// TIA Portal project "Buffer" (V18)

(* hardware
DEVICE "S7-1500/ET200MP station_1"  S7-1500 station
   slot 0: "Rail_0"  Rack  6ES7 590-1***0-0AA0
   slot 1: "PLC_1"  CPU 1515-2 PN  6ES7 515-2AN03-0AB0  V3.0
      slot 3: "CPU display_1"  6ES7591-1BA00-0AA0
      slot 32768: "PROFINET interface_1"  X1
         slot 32769: "Port_1"  X1 P1
         slot 32770: "Port_2"  X1 P2
      slot 33024: "PROFINET interface_2"  X2
         slot 33025: "Port_1"  X2 P1
      slot 34817: "Virtual CP interface port_1"  Virtual CP interface port  Virtual CP interface port
*)

// ===== PLC "PLC_1"  CPU 1515-2 PN =====

VAR_GLOBAL   // PLC tag table "Default tag table"
   "System_Byte" AT %MB0 : Byte;
   "FirstScan" AT %M0.0 : Bool;
   "DiagStatusUpdate" AT %M0.1 : Bool;
   "AlwaysTRUE" AT %M0.2 : Bool;
   "AlwaysFALSE" AT %M0.3 : Bool;
   "Clock_Byte" AT %MB1 : Byte;
   "Clock_10Hz" AT %M1.0 : Bool;
   "Clock_5Hz" AT %M1.1 : Bool;
   "Clock_2.5Hz" AT %M1.2 : Bool;
   "Clock_2Hz" AT %M1.3 : Bool;
   "Clock_1.25Hz" AT %M1.4 : Bool;
   "Clock_1Hz" AT %M1.5 : Bool;
   "Clock_0.625Hz" AT %M1.6 : Bool;
   "Clock_0.5Hz" AT %M1.7 : Bool;
   "Index" AT %MD18 : UDInt;
   "Start" AT %M16.0 : Bool;
   "Start2" AT %M16.1 : Bool;
   "FoundIndex" AT %MW20 : Word;
   "Tag_1" AT %M16.2 : Bool;
   "Tag_2" AT %MW22 : Int;
END_VAR

VAR_GLOBAL CONSTANT   // PLC tag table "Default tag table"
   "c_MAX_RECORD_LEN" : Int := 100;   // //Max length of single record [Byte]
END_VAR

TYPE "udt_DATABASE3"
   STRUCT
      FirstName : Array[1..10] of Char;
      Lastname : Array[1..20] of Char;
      Age : USInt;
      Details : Struct
         Male : Bool;
         COMPLETE_TO_WORD2 : Bool;
         COMPLETE_TO_WORD3 : Bool;
         COMPLETE_TO_WORD4 : Bool;
         COMPLETE_TO_WORD5 : Bool;
         COMPLETE_TO_WORD6 : Bool;
         COMPLETE_TO_WORD7 : Bool;
         COMPLETE_TO_WORD8 : Bool;
         COMPLETE_TO_WORD9 : Bool;
         COMPLETE_TO_WORD10 : Bool;
         COMPLETE_TO_WORD11 : Bool;
         COMPLETE_TO_WORD12 : Bool;
         COMPLETE_TO_WORD13 : Bool;
         COMPLETE_TO_WORD14 : Bool;
         COMPLETE_TO_WORD15 : Bool;
         COMPLETE_TO_WORD16 : Bool;
      END_STRUCT;
   END_STRUCT;
END_TYPE

// folder: DATABASES

DATA_BLOCK "db_DATABASE_1"   // DB100
{ S7_Optimized_Access := 'TRUE' }
VERSION : 0.1
   VAR
      Act_Records : UDInt;
      WorkRecord : Byte;
      RecordMask : Byte;
      Database : Array[1..1000] of Byte;
   END_VAR
BEGIN
END_DATA_BLOCK

DATA_BLOCK "db_DATABASE_2"   // DB101
{ S7_Optimized_Access := 'TRUE' }
VERSION : 0.1
   VAR
      Act_Records : UDInt;
      WorkRecord : Real;
      RecordMask : Real;
      Database : Array[1..1000] of Real;
   END_VAR
BEGIN
END_DATA_BLOCK

DATA_BLOCK "db_DATABASE_3"   // DB102
{ S7_Optimized_Access := 'TRUE' }
VERSION : 0.1
   VAR
      Act_Records : UDInt;
      WorkRecord : "udt_DATABASE3";
      RecordMask : "udt_DATABASE3";
      Database : Array[1..1000] of "udt_DATABASE3";
   END_VAR
BEGIN
END_DATA_BLOCK

// folder: DB_TOOLS

DATA_BLOCK "db_Records"   // DB1
{ S7_Optimized_Access := 'TRUE' }
VERSION : 0.1
   VAR
      Push : Struct
         Record1 : Byte;
         Record2 : Real;
         Record3 : "udt_DATABASE3";
      END_STRUCT;
      Pop : Struct
         Record1 : Byte;
         Record2 : Real;
         Record3 : "udt_DATABASE3";
      END_STRUCT;
      Shift : Struct
         Record1 : Byte;
         Record2 : Real;
         Record3 : "udt_DATABASE3";
      END_STRUCT;
      Unshift : Struct
         Record1 : Byte;
         Record2 : Real;
         Record3 : "udt_DATABASE3";
      END_STRUCT;
      Insert : Struct
         Record1 : Byte;
         Record2 : Real;
         Record3 : "udt_DATABASE3";
      END_STRUCT;
      Remove : Struct
         Record1 : Byte;
         Record2 : Real;
         Record3 : "udt_DATABASE3";
      END_STRUCT;
      Read : Struct
         Record1 : Byte;
         Record2 : Real;
         Record3 : "udt_DATABASE3";
      END_STRUCT;
      ReadLast : Struct
         Record1 : Byte;
         Record2 : Real;
         Record3 : "udt_DATABASE3";
      END_STRUCT;
      Overwrite : Struct
         Record1 : Byte;
         Record2 : Real;
         Record3 : "udt_DATABASE3";
      END_STRUCT;
      OverwriteLast : Struct
         Record1 : Byte;
         Record2 : Real;
         Record3 : "udt_DATABASE3";
      END_STRUCT;
      Find : Struct
         Record1 : Byte;
         Record2 : Real;
         Record3 : "udt_DATABASE3";
      END_STRUCT;
   END_VAR
BEGIN
END_DATA_BLOCK

// folder: (top level)

FUNCTION "fc_PushCall" : Void   // FC1, LAD
{ S7_Optimized_Access := 'TRUE' }
VERSION : 0.1
   VAR_TEMP
      _DONE : Bool;
   END_VAR
BEGIN

REGION Network 1: Push into Database 1
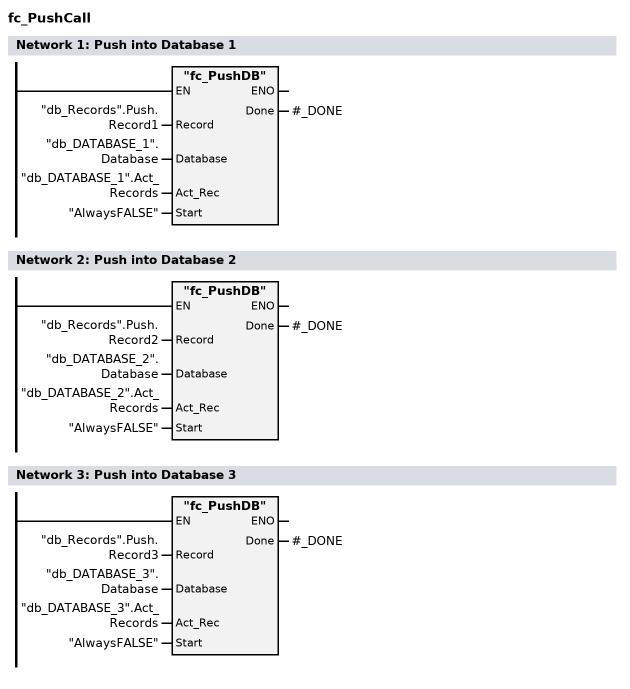
   RUNG wire#powerrail
      "fc_PushDB"(Record := "db_Records".Push.Record1, Database := "db_DATABASE_1".Database, Act_Rec := "db_DATABASE_1".Act_Records, Start := "AlwaysFALSE", Done => #_DONE)
   END_RUNG
   // the same network as SCL:
   "fc_PushDB"(Record := "db_Records".Push.Record1,
               Database := "db_DATABASE_1".Database,
               Act_Rec := "db_DATABASE_1".Act_Records,
               Start := "AlwaysFALSE",
               Done => #_DONE);
END_REGION

REGION Network 2: Push into Database 2
   RUNG wire#powerrail
      "fc_PushDB"(Record := "db_Records".Push.Record2, Database := "db_DATABASE_2".Database, Act_Rec := "db_DATABASE_2".Act_Records, Start := "AlwaysFALSE", Done => #_DONE)
   END_RUNG
   // the same network as SCL:
   "fc_PushDB"(Record := "db_Records".Push.Record2,
               Database := "db_DATABASE_2".Database,
               Act_Rec := "db_DATABASE_2".Act_Records,
               Start := "AlwaysFALSE",
               Done => #_DONE);
END_REGION

REGION Network 3: Push into Database 3
   RUNG wire#powerrail
      "fc_PushDB"(Record := "db_Records".Push.Record3, Database := "db_DATABASE_3".Database, Act_Rec := "db_DATABASE_3".Act_Records, Start := "AlwaysFALSE", Done => #_DONE)
   END_RUNG
   // the same network as SCL:
   "fc_PushDB"(Record := "db_Records".Push.Record3,
               Database := "db_DATABASE_3".Database,
               Act_Rec := "db_DATABASE_3".Act_Records,
               Start := "AlwaysFALSE",
               Done => #_DONE);
END_REGION
END_FUNCTION

FUNCTION "fc_PopCall" : Void   // FC2, LAD
{ S7_Optimized_Access := 'TRUE' }
VERSION : 0.1
   VAR_TEMP
      _DONE : Bool;
   END_VAR
BEGIN

REGION Network 1: Pop from Database 1
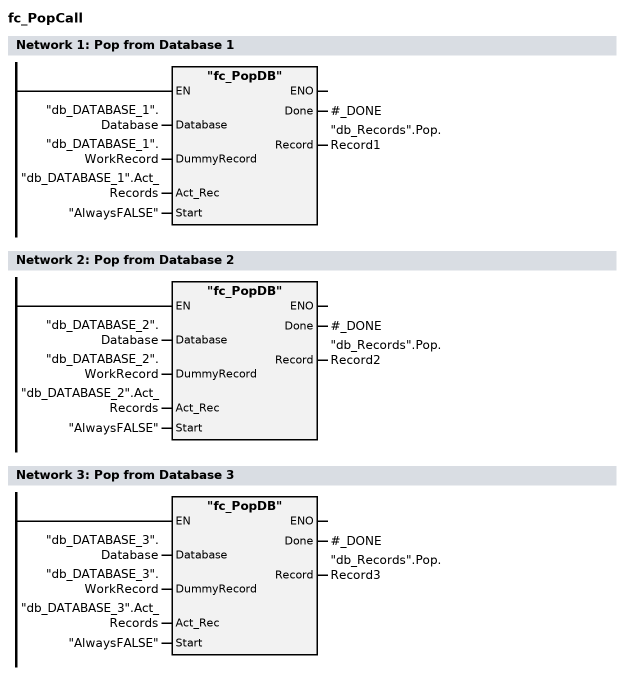
   RUNG wire#powerrail
      "fc_PopDB"(Database := "db_DATABASE_1".Database, DummyRecord := "db_DATABASE_1".WorkRecord, Act_Rec := "db_DATABASE_1".Act_Records, Start := "AlwaysFALSE", Done => #_DONE, Record => "db_Records".Pop.Record1)
   END_RUNG
   // the same network as SCL:
   "fc_PopDB"(Database := "db_DATABASE_1".Database,
              DummyRecord := "db_DATABASE_1".WorkRecord,
              Act_Rec := "db_DATABASE_1".Act_Records,
              Start := "AlwaysFALSE",
              Done => #_DONE,
              Record => "db_Records".Pop.Record1);
END_REGION

REGION Network 2: Pop from Database 2
   RUNG wire#powerrail
      "fc_PopDB"(Database := "db_DATABASE_2".Database, DummyRecord := "db_DATABASE_2".WorkRecord, Act_Rec := "db_DATABASE_2".Act_Records, Start := "AlwaysFALSE", Done => #_DONE, Record => "db_Records".Pop.Record2)
   END_RUNG
   // the same network as SCL:
   "fc_PopDB"(Database := "db_DATABASE_2".Database,
              DummyRecord := "db_DATABASE_2".WorkRecord,
              Act_Rec := "db_DATABASE_2".Act_Records,
              Start := "AlwaysFALSE",
              Done => #_DONE,
              Record => "db_Records".Pop.Record2);
END_REGION

REGION Network 3: Pop from Database 3
   RUNG wire#powerrail
      "fc_PopDB"(Database := "db_DATABASE_3".Database, DummyRecord := "db_DATABASE_3".WorkRecord, Act_Rec := "db_DATABASE_3".Act_Records, Start := "AlwaysFALSE", Done => #_DONE, Record => "db_Records".Pop.Record3)
   END_RUNG
   // the same network as SCL:
   "fc_PopDB"(Database := "db_DATABASE_3".Database,
              DummyRecord := "db_DATABASE_3".WorkRecord,
              Act_Rec := "db_DATABASE_3".Act_Records,
              Start := "AlwaysFALSE",
              Done => #_DONE,
              Record => "db_Records".Pop.Record3);
END_REGION
END_FUNCTION

FUNCTION "fc_ShiftCall" : Void   // FC3, LAD
{ S7_Optimized_Access := 'TRUE' }
VERSION : 0.1
   VAR_TEMP
      _DONE : Bool;
   END_VAR
BEGIN

REGION Network 1: Shift from Database 1
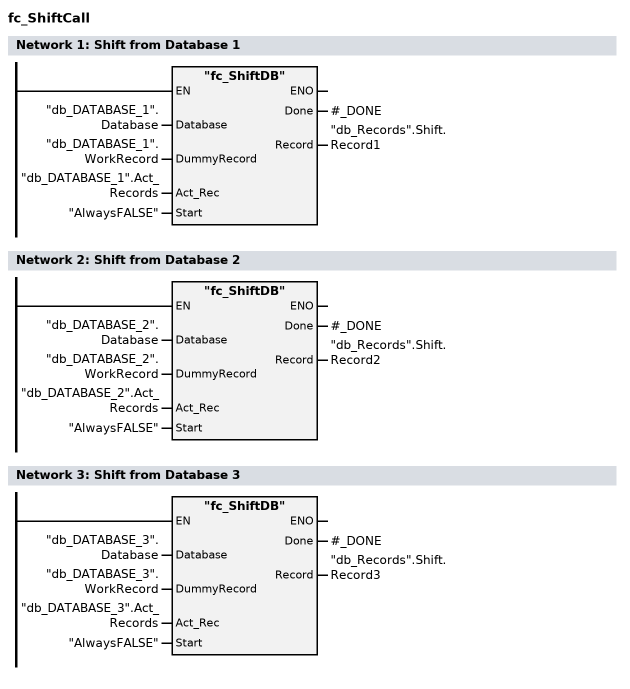
   RUNG wire#powerrail
      "fc_ShiftDB"(Record => "db_Records".Shift.Record1, Database := "db_DATABASE_1".Database, DummyRecord := "db_DATABASE_1".WorkRecord, Act_Rec := "db_DATABASE_1".Act_Records, Start := "AlwaysFALSE", Done => #_DONE)
   END_RUNG
   // the same network as SCL:
   "fc_ShiftDB"(Database := "db_DATABASE_1".Database,
                DummyRecord := "db_DATABASE_1".WorkRecord,
                Act_Rec := "db_DATABASE_1".Act_Records,
                Start := "AlwaysFALSE",
                Done => #_DONE,
                Record => "db_Records".Shift.Record1);
END_REGION

REGION Network 2: Shift from Database 2
   RUNG wire#powerrail
      "fc_ShiftDB"(Record => "db_Records".Shift.Record2, Database := "db_DATABASE_2".Database, DummyRecord := "db_DATABASE_2".WorkRecord, Act_Rec := "db_DATABASE_2".Act_Records, Start := "AlwaysFALSE", Done => #_DONE)
   END_RUNG
   // the same network as SCL:
   "fc_ShiftDB"(Database := "db_DATABASE_2".Database,
                DummyRecord := "db_DATABASE_2".WorkRecord,
                Act_Rec := "db_DATABASE_2".Act_Records,
                Start := "AlwaysFALSE",
                Done => #_DONE,
                Record => "db_Records".Shift.Record2);
END_REGION

REGION Network 3: Shift from Database 3
   RUNG wire#powerrail
      "fc_ShiftDB"(Record => "db_Records".Shift.Record3, Database := "db_DATABASE_3".Database, DummyRecord := "db_DATABASE_3".WorkRecord, Act_Rec := "db_DATABASE_3".Act_Records, Start := "AlwaysFALSE", Done => #_DONE)
   END_RUNG
   // the same network as SCL:
   "fc_ShiftDB"(Database := "db_DATABASE_3".Database,
                DummyRecord := "db_DATABASE_3".WorkRecord,
                Act_Rec := "db_DATABASE_3".Act_Records,
                Start := "AlwaysFALSE",
                Done => #_DONE,
                Record => "db_Records".Shift.Record3);
END_REGION
END_FUNCTION

FUNCTION "fc_UnshiftCall" : Void   // FC4, LAD
{ S7_Optimized_Access := 'TRUE' }
VERSION : 0.1
   VAR_TEMP
      _DONE : Bool;
   END_VAR
BEGIN

REGION Network 1: Unshift into Database 1
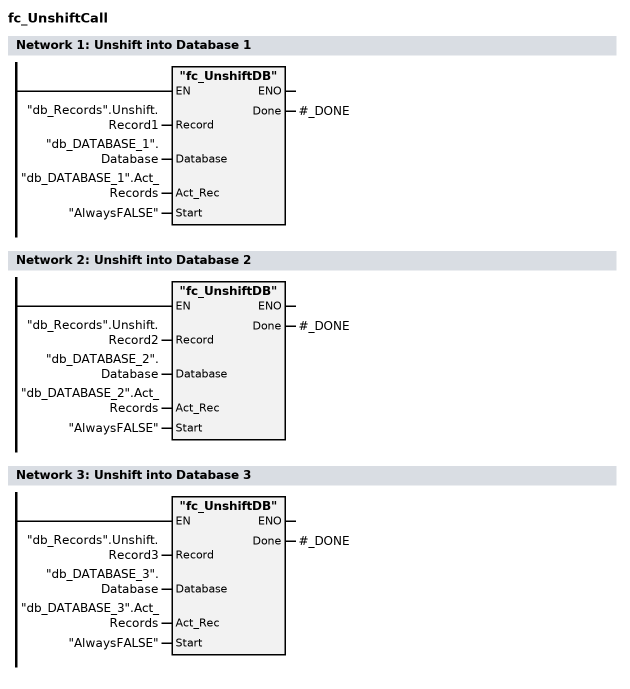
   RUNG wire#powerrail
      "fc_UnshiftDB"(Record := "db_Records".Unshift.Record1, Database := "db_DATABASE_1".Database, Act_Rec := "db_DATABASE_1".Act_Records, Start := "AlwaysFALSE", Done => #_DONE)
   END_RUNG
   // the same network as SCL:
   "fc_UnshiftDB"(Record := "db_Records".Unshift.Record1,
                  Database := "db_DATABASE_1".Database,
                  Act_Rec := "db_DATABASE_1".Act_Records,
                  Start := "AlwaysFALSE",
                  Done => #_DONE);
END_REGION

REGION Network 2: Unshift into Database 2
   RUNG wire#powerrail
      "fc_UnshiftDB"(Record := "db_Records".Unshift.Record2, Database := "db_DATABASE_2".Database, Act_Rec := "db_DATABASE_2".Act_Records, Start := "AlwaysFALSE", Done => #_DONE)
   END_RUNG
   // the same network as SCL:
   "fc_UnshiftDB"(Record := "db_Records".Unshift.Record2,
                  Database := "db_DATABASE_2".Database,
                  Act_Rec := "db_DATABASE_2".Act_Records,
                  Start := "AlwaysFALSE",
                  Done => #_DONE);
END_REGION

REGION Network 3: Unshift into Database 3
   RUNG wire#powerrail
      "fc_UnshiftDB"(Record := "db_Records".Unshift.Record3, Database := "db_DATABASE_3".Database, Act_Rec := "db_DATABASE_3".Act_Records, Start := "AlwaysFALSE", Done => #_DONE)
   END_RUNG
   // the same network as SCL:
   "fc_UnshiftDB"(Record := "db_Records".Unshift.Record3,
                  Database := "db_DATABASE_3".Database,
                  Act_Rec := "db_DATABASE_3".Act_Records,
                  Start := "AlwaysFALSE",
                  Done => #_DONE);
END_REGION
END_FUNCTION

FUNCTION "fc_ClearCall" : Void   // FC5, LAD
{ S7_Optimized_Access := 'TRUE' }
VERSION : 0.1
   VAR_TEMP
      _DONE : Bool;
   END_VAR
BEGIN

REGION Network 1: Clear Database 1
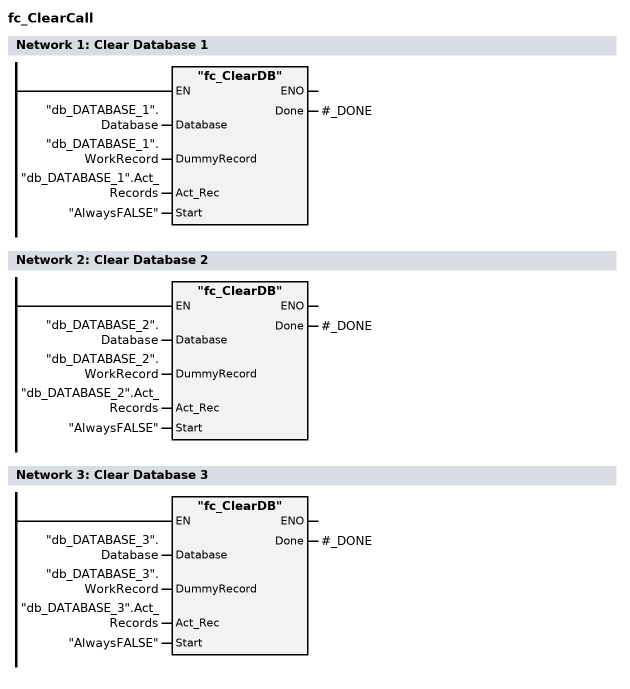
   RUNG wire#powerrail
      "fc_ClearDB"(Database := "db_DATABASE_1".Database, DummyRecord := "db_DATABASE_1".WorkRecord, Act_Rec := "db_DATABASE_1".Act_Records, Start := "AlwaysFALSE", Done => #_DONE)
   END_RUNG
   // the same network as SCL:
   "fc_ClearDB"(Database := "db_DATABASE_1".Database,
                DummyRecord := "db_DATABASE_1".WorkRecord,
                Act_Rec := "db_DATABASE_1".Act_Records,
                Start := "AlwaysFALSE",
                Done => #_DONE);
END_REGION

REGION Network 2: Clear Database 2
   RUNG wire#powerrail
      "fc_ClearDB"(Database := "db_DATABASE_2".Database, DummyRecord := "db_DATABASE_2".WorkRecord, Act_Rec := "db_DATABASE_2".Act_Records, Start := "AlwaysFALSE", Done => #_DONE)
   END_RUNG
   // the same network as SCL:
   "fc_ClearDB"(Database := "db_DATABASE_2".Database,
                DummyRecord := "db_DATABASE_2".WorkRecord,
                Act_Rec := "db_DATABASE_2".Act_Records,
                Start := "AlwaysFALSE",
                Done => #_DONE);
END_REGION

REGION Network 3: Clear Database 3
   RUNG wire#powerrail
      "fc_ClearDB"(Database := "db_DATABASE_3".Database, DummyRecord := "db_DATABASE_3".WorkRecord, Act_Rec := "db_DATABASE_3".Act_Records, Start := "AlwaysFALSE", Done => #_DONE)
   END_RUNG
   // the same network as SCL:
   "fc_ClearDB"(Database := "db_DATABASE_3".Database,
                DummyRecord := "db_DATABASE_3".WorkRecord,
                Act_Rec := "db_DATABASE_3".Act_Records,
                Start := "AlwaysFALSE",
                Done => #_DONE);
END_REGION
END_FUNCTION

FUNCTION "fc_InsertCall" : Void   // FC6, LAD
{ S7_Optimized_Access := 'TRUE' }
VERSION : 0.1
   VAR_TEMP
      _DONE : Bool;
   END_VAR
BEGIN

REGION Network 1: Insert into Database 1
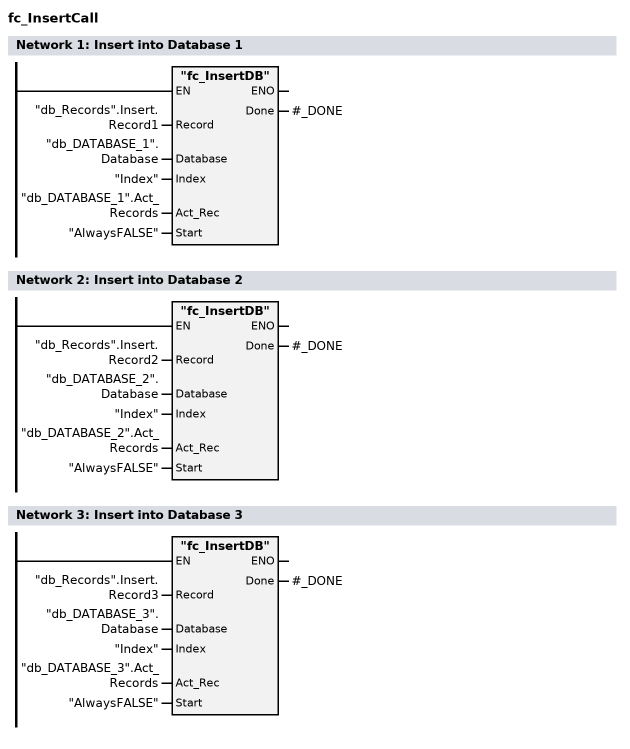
   RUNG wire#powerrail
      "fc_InsertDB"(Record := "db_Records".Insert.Record1, Database := "db_DATABASE_1".Database, Index := "Index", Act_Rec := "db_DATABASE_1".Act_Records, Start := "AlwaysFALSE", Done => #_DONE)
   END_RUNG
   // the same network as SCL:
   "fc_InsertDB"(Record := "db_Records".Insert.Record1,
                 Database := "db_DATABASE_1".Database,
                 Index := "Index",
                 Act_Rec := "db_DATABASE_1".Act_Records,
                 Start := "AlwaysFALSE",
                 Done => #_DONE);
END_REGION

REGION Network 2: Insert into Database 2
   RUNG wire#powerrail
      "fc_InsertDB"(Record := "db_Records".Insert.Record2, Database := "db_DATABASE_2".Database, Index := "Index", Act_Rec := "db_DATABASE_2".Act_Records, Start := "AlwaysFALSE", Done => #_DONE)
   END_RUNG
   // the same network as SCL:
   "fc_InsertDB"(Record := "db_Records".Insert.Record2,
                 Database := "db_DATABASE_2".Database,
                 Index := "Index",
                 Act_Rec := "db_DATABASE_2".Act_Records,
                 Start := "AlwaysFALSE",
                 Done => #_DONE);
END_REGION

REGION Network 3: Insert into Database 3
   RUNG wire#powerrail
      "fc_InsertDB"(Record := "db_Records".Insert.Record3, Database := "db_DATABASE_3".Database, Index := "Index", Act_Rec := "db_DATABASE_3".Act_Records, Start := "AlwaysFALSE", Done => #_DONE)
   END_RUNG
   // the same network as SCL:
   "fc_InsertDB"(Record := "db_Records".Insert.Record3,
                 Database := "db_DATABASE_3".Database,
                 Index := "Index",
                 Act_Rec := "db_DATABASE_3".Act_Records,
                 Start := "AlwaysFALSE",
                 Done => #_DONE);
END_REGION
END_FUNCTION

FUNCTION "fc_RemoveCall" : Void   // FC7, LAD
{ S7_Optimized_Access := 'TRUE' }
VERSION : 0.1
   VAR_TEMP
      _DONE : Bool;
   END_VAR
BEGIN

REGION Network 1: Remove from Database 1
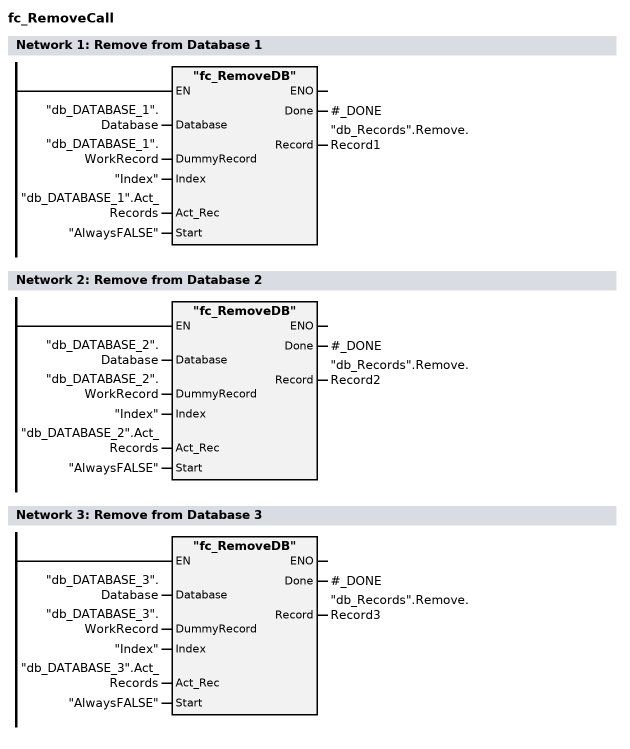
   RUNG wire#powerrail
      "fc_RemoveDB"(Database := "db_DATABASE_1".Database, DummyRecord := "db_DATABASE_1".WorkRecord, Index := "Index", Act_Rec := "db_DATABASE_1".Act_Records, Start := "AlwaysFALSE", Done => #_DONE, Record => "db_Records".Remove.Record1)
   END_RUNG
   // the same network as SCL:
   "fc_RemoveDB"(Database := "db_DATABASE_1".Database,
                 DummyRecord := "db_DATABASE_1".WorkRecord,
                 Index := "Index",
                 Act_Rec := "db_DATABASE_1".Act_Records,
                 Start := "AlwaysFALSE",
                 Done => #_DONE,
                 Record => "db_Records".Remove.Record1);
END_REGION

REGION Network 2: Remove from Database 2
   RUNG wire#powerrail
      "fc_RemoveDB"(Database := "db_DATABASE_2".Database, DummyRecord := "db_DATABASE_2".WorkRecord, Index := "Index", Act_Rec := "db_DATABASE_2".Act_Records, Start := "AlwaysFALSE", Done => #_DONE, Record => "db_Records".Remove.Record2)
   END_RUNG
   // the same network as SCL:
   "fc_RemoveDB"(Database := "db_DATABASE_2".Database,
                 DummyRecord := "db_DATABASE_2".WorkRecord,
                 Index := "Index",
                 Act_Rec := "db_DATABASE_2".Act_Records,
                 Start := "AlwaysFALSE",
                 Done => #_DONE,
                 Record => "db_Records".Remove.Record2);
END_REGION

REGION Network 3: Remove from Database 3
   RUNG wire#powerrail
      "fc_RemoveDB"(Database := "db_DATABASE_3".Database, DummyRecord := "db_DATABASE_3".WorkRecord, Index := "Index", Act_Rec := "db_DATABASE_3".Act_Records, Start := "AlwaysFALSE", Done => #_DONE, Record => "db_Records".Remove.Record3)
   END_RUNG
   // the same network as SCL:
   "fc_RemoveDB"(Database := "db_DATABASE_3".Database,
                 DummyRecord := "db_DATABASE_3".WorkRecord,
                 Index := "Index",
                 Act_Rec := "db_DATABASE_3".Act_Records,
                 Start := "AlwaysFALSE",
                 Done => #_DONE,
                 Record => "db_Records".Remove.Record3);
END_REGION
END_FUNCTION

FUNCTION "fc_ReadCall" : Void   // FC8, LAD
{ S7_Optimized_Access := 'TRUE' }
VERSION : 0.1
   VAR_TEMP
      _DONE : Bool;
   END_VAR
BEGIN

REGION Network 1: Read from Database 1
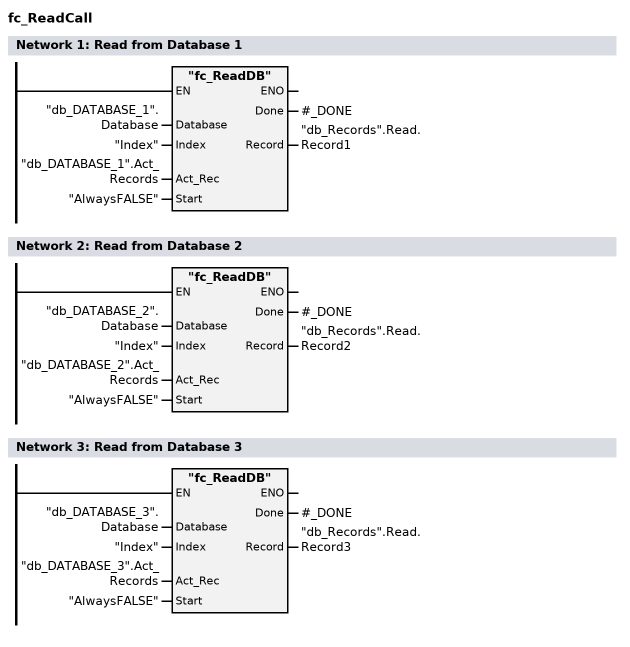
   RUNG wire#powerrail
      "fc_ReadDB"(Record => "db_Records".Read.Record1, Database := "db_DATABASE_1".Database, Index := "Index", Act_Rec := "db_DATABASE_1".Act_Records, Start := "AlwaysFALSE", Done => #_DONE)
   END_RUNG
   // the same network as SCL:
   "fc_ReadDB"(Database := "db_DATABASE_1".Database,
               Index := "Index",
               Act_Rec := "db_DATABASE_1".Act_Records,
               Start := "AlwaysFALSE",
               Done => #_DONE,
               Record => "db_Records".Read.Record1);
END_REGION

REGION Network 2: Read from Database 2
   RUNG wire#powerrail
      "fc_ReadDB"(Record => "db_Records".Read.Record2, Database := "db_DATABASE_2".Database, Index := "Index", Act_Rec := "db_DATABASE_2".Act_Records, Start := "AlwaysFALSE", Done => #_DONE)
   END_RUNG
   // the same network as SCL:
   "fc_ReadDB"(Database := "db_DATABASE_2".Database,
               Index := "Index",
               Act_Rec := "db_DATABASE_2".Act_Records,
               Start := "AlwaysFALSE",
               Done => #_DONE,
               Record => "db_Records".Read.Record2);
END_REGION

REGION Network 3: Read from Database 3
   RUNG wire#powerrail
      "fc_ReadDB"(Record => "db_Records".Read.Record3, Database := "db_DATABASE_3".Database, Index := "Index", Act_Rec := "db_DATABASE_3".Act_Records, Start := "AlwaysFALSE", Done => #_DONE)
   END_RUNG
   // the same network as SCL:
   "fc_ReadDB"(Database := "db_DATABASE_3".Database,
               Index := "Index",
               Act_Rec := "db_DATABASE_3".Act_Records,
               Start := "AlwaysFALSE",
               Done => #_DONE,
               Record => "db_Records".Read.Record3);
END_REGION
END_FUNCTION

FUNCTION "fc_ReadLastCall" : Void   // FC9, LAD
{ S7_Optimized_Access := 'TRUE' }
VERSION : 0.1
   VAR_TEMP
      _DONE : Bool;
   END_VAR
BEGIN

REGION Network 1: Read last from Database 1
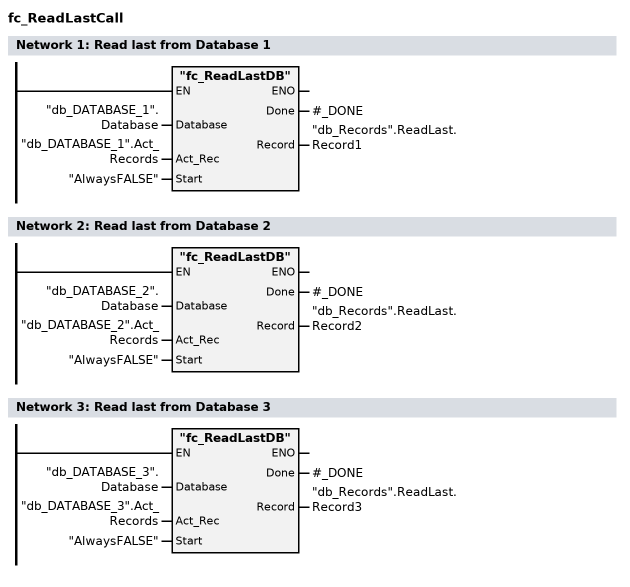
   RUNG wire#powerrail
      "fc_ReadLastDB"(Database := "db_DATABASE_1".Database, Act_Rec := "db_DATABASE_1".Act_Records, Start := "AlwaysFALSE", Done => #_DONE, Record => "db_Records".ReadLast.Record1)
   END_RUNG
   // the same network as SCL:
   "fc_ReadLastDB"(Database := "db_DATABASE_1".Database,
                   Act_Rec := "db_DATABASE_1".Act_Records,
                   Start := "AlwaysFALSE",
                   Done => #_DONE,
                   Record => "db_Records".ReadLast.Record1);
END_REGION

REGION Network 2: Read last from Database 2
   RUNG wire#powerrail
      "fc_ReadLastDB"(Database := "db_DATABASE_2".Database, Act_Rec := "db_DATABASE_2".Act_Records, Start := "AlwaysFALSE", Done => #_DONE, Record => "db_Records".ReadLast.Record2)
   END_RUNG
   // the same network as SCL:
   "fc_ReadLastDB"(Database := "db_DATABASE_2".Database,
                   Act_Rec := "db_DATABASE_2".Act_Records,
                   Start := "AlwaysFALSE",
                   Done => #_DONE,
                   Record => "db_Records".ReadLast.Record2);
END_REGION

REGION Network 3: Read last from Database 3
   RUNG wire#powerrail
      "fc_ReadLastDB"(Database := "db_DATABASE_3".Database, Act_Rec := "db_DATABASE_3".Act_Records, Start := "AlwaysFALSE", Done => #_DONE, Record => "db_Records".ReadLast.Record3)
   END_RUNG
   // the same network as SCL:
   "fc_ReadLastDB"(Database := "db_DATABASE_3".Database,
                   Act_Rec := "db_DATABASE_3".Act_Records,
                   Start := "AlwaysFALSE",
                   Done => #_DONE,
                   Record => "db_Records".ReadLast.Record3);
END_REGION
END_FUNCTION

FUNCTION "fc_FindCall" : Void   // FC12, LAD
{ S7_Optimized_Access := 'TRUE' }
VERSION : 0.1
   VAR_TEMP
      _FOUND : Bool;
      _DONE : Bool;
      _INDEX : UDInt;
      _FILL : Byte;
   END_VAR
   VAR_TEMP   // added for the SCL form of the ladder/FBD networks
      _w1 : Bool;
   END_VAR
BEGIN

REGION Network 1 (STL)
         L     16#0;
         T     #_FILL;
END_REGION

REGION Network 2 (STL): Create RecordMask for Database 1
         CALL  "fc_FILL_STRUCT"
         ( ByVAL    := #_FILL,
           "Struct" := "db_DATABASE_1".RecordMask
         );

         L     16#FF;
         T     "db_DATABASE_1".RecordMask;
END_REGION

REGION Network 3: Find in Database 1
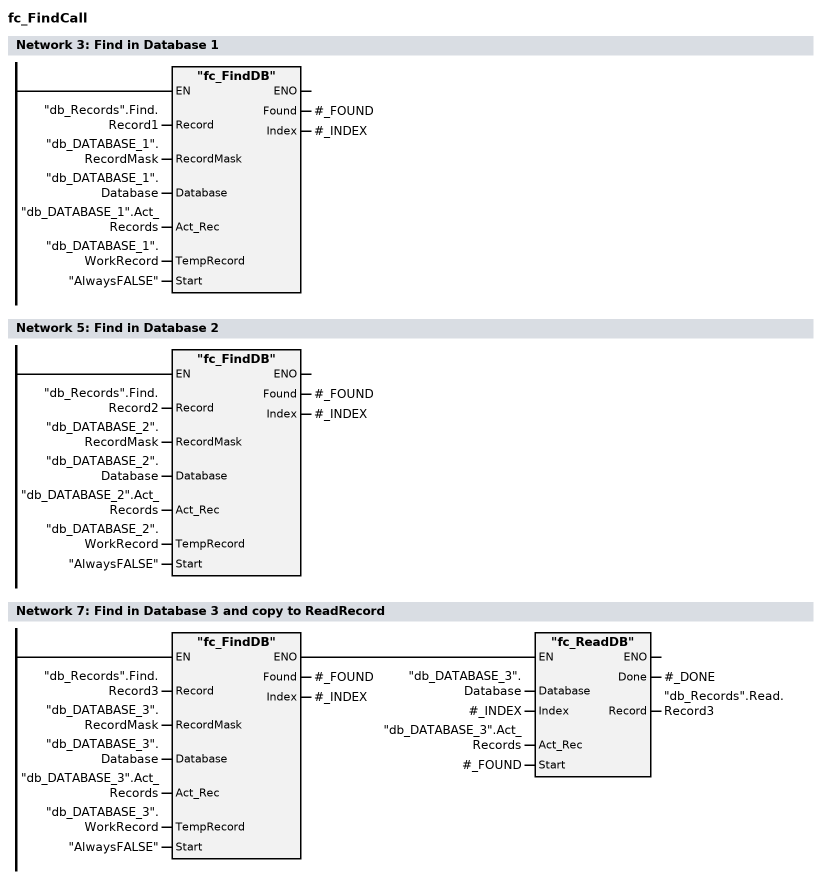
   RUNG wire#powerrail
      "fc_FindDB"(Record := "db_Records".Find.Record1, RecordMask := "db_DATABASE_1".RecordMask, Database := "db_DATABASE_1".Database, Start := "AlwaysFALSE", Act_Rec := "db_DATABASE_1".Act_Records, TempRecord := "db_DATABASE_1".WorkRecord, Found => #_FOUND, Index => #_INDEX)
   END_RUNG
   // the same network as SCL:
   "fc_FindDB"(Record := "db_Records".Find.Record1,
               RecordMask := "db_DATABASE_1".RecordMask,
               Database := "db_DATABASE_1".Database,
               Act_Rec := "db_DATABASE_1".Act_Records,
               TempRecord := "db_DATABASE_1".WorkRecord,
               Start := "AlwaysFALSE",
               Found => #_FOUND,
               Index => #_INDEX);
END_REGION

REGION Network 4 (STL): Create RecordMask for Database 2
         CALL  "fc_FILL_STRUCT"
         ( ByVAL    := #_FILL,
           "Struct" := "db_DATABASE_2".RecordMask
         );

         L     16#FFFFFFFF;
         T     "db_DATABASE_2".RecordMask;
END_REGION

REGION Network 5: Find in Database 2
   RUNG wire#powerrail
      "fc_FindDB"(Record := "db_Records".Find.Record2, RecordMask := "db_DATABASE_2".RecordMask, Database := "db_DATABASE_2".Database, Start := "AlwaysFALSE", Act_Rec := "db_DATABASE_2".Act_Records, TempRecord := "db_DATABASE_2".WorkRecord, Found => #_FOUND, Index => #_INDEX)
   END_RUNG
   // the same network as SCL:
   "fc_FindDB"(Record := "db_Records".Find.Record2,
               RecordMask := "db_DATABASE_2".RecordMask,
               Database := "db_DATABASE_2".Database,
               Act_Rec := "db_DATABASE_2".Act_Records,
               TempRecord := "db_DATABASE_2".WorkRecord,
               Start := "AlwaysFALSE",
               Found => #_FOUND,
               Index => #_INDEX);
END_REGION

REGION Network 6 (STL): Create RecordMask for Database 3
         CALL  "fc_FILL_STRUCT"
         ( ByVAL    := #_FILL,
           "Struct" := "db_DATABASE_3".RecordMask
         );

   //Znajdz pierwszy rekord, ktory ma okreslona ilosc lat (Age)
   //L     16#FF
   //T     "db_DATABASE_3".RecordMask.FirstName[1]
   //T     "db_DATABASE_3".RecordMask.FirstName[2]
   //T     "db_DATABASE_3".RecordMask.FirstName[3]
   //T     "db_DATABASE_3".RecordMask.FirstName[4]
   //T     "db_DATABASE_3".RecordMask.FirstName[5]
   //T     "db_DATABASE_3".RecordMask.FirstName[6]
   //T     "db_DATABASE_3".RecordMask.FirstName[7]
   //T     "db_DATABASE_3".RecordMask.FirstName[8]
   //T     "db_DATABASE_3".RecordMask.FirstName[9]
   //T     "db_DATABASE_3".RecordMask.FirstName[10]

   //Znajdz pierwszy rekord, ktory ma okreslana plec (Male)
         CALL  "fc_FILL_STRUCT"
         ( ByVAL    := 16#FF,
           "Struct" := "db_DATABASE_3".RecordMask.Lastname
         );
END_REGION

REGION Network 7: Find in Database 3 and copy to ReadRecord
   RUNG wire#powerrail
      "fc_FindDB"(Record := "db_Records".Find.Record3, RecordMask := "db_DATABASE_3".RecordMask, Database := "db_DATABASE_3".Database, Act_Rec := "db_DATABASE_3".Act_Records, TempRecord := "db_DATABASE_3".WorkRecord, Start := "AlwaysFALSE", Found => #_FOUND, Index => #_INDEX)
      "fc_ReadDB"(Database := "db_DATABASE_3".Database, Index := #_INDEX, Act_Rec := "db_DATABASE_3".Act_Records, Start := #_FOUND, Done => #_DONE, Record => "db_Records".Read.Record3)
   END_RUNG
   // the same network as SCL:
   "fc_FindDB"(Record := "db_Records".Find.Record3,
               RecordMask := "db_DATABASE_3".RecordMask,
               Database := "db_DATABASE_3".Database,
               Act_Rec := "db_DATABASE_3".Act_Records,
               TempRecord := "db_DATABASE_3".WorkRecord,
               Start := "AlwaysFALSE",
               Found => #_FOUND,
               Index => #_INDEX,
               ENO => #_w1);
   IF #_w1 THEN
       "fc_ReadDB"(Database := "db_DATABASE_3".Database,
                   Index := #_INDEX,
                   Act_Rec := "db_DATABASE_3".Act_Records,
                   Start := #_FOUND,
                   Done => #_DONE,
                   Record => "db_Records".Read.Record3);
   END_IF;
END_REGION
END_FUNCTION

ORGANIZATION_BLOCK "Main"   // OB1, LAD, ProgramCycle
TITLE = "Main Program Sweep (Cycle)"
{ S7_Optimized_Access := 'TRUE' }
VERSION : 0.1
   VAR_INPUT
      Initial_Call : Bool;   // Initial call of this OB
      Remanence : Bool;   // =True, if remanent data are available
   END_VAR
BEGIN

REGION Network 1 (STL): Databases
         CALL  "fc_PushCall";
         CALL  "fc_PopCall";
         CALL  "fc_ShiftCall";
         CALL  "fc_UnshiftCall";
         CALL  "fc_ClearCall";
         CALL  "fc_InsertCall";
         CALL  "fc_RemoveCall";
         CALL  "fc_ReadCall";
         CALL  "fc_ReadLastCall";
         CALL  "fc_FindCall";
END_REGION
END_ORGANIZATION_BLOCK

// folder: DB_TOOLS

FUNCTION "fc_PushDB" : Void   // FC111, SCL
{ S7_Optimized_Access := 'TRUE' }
VERSION : 0.1
   VAR_INPUT
      Record : Variant;
      Database : Variant;
   END_VAR
   VAR_OUTPUT
      Done : Bool;
   END_VAR
   VAR_IN_OUT
      Act_Rec : UDInt;
      Start : Bool;
   END_VAR
   VAR_TEMP
      _CountElements : UDInt;
      _RetVal : Int;
      _DummyByte : Byte;
      _DummyArray : Array[1..1000] of Byte;
   END_VAR
BEGIN
   REGION NOT #Done
       #Done := FALSE;
   END_REGION

   REGION #Start
       IF #Start THEN
           #Start := FALSE;
       ELSE
           RETURN;
       END_IF;
   END_REGION

   REGION Check Database
       IF IS_ARRAY(#Database) THEN
           #_CountElements := CountOfElements(#Database);
       ELSE
           RETURN;
       END_IF;
       IF #Act_Rec >= #_CountElements THEN
           RETURN;
       END_IF;
   END_REGION

   REGION Check Record
       IF TypeOf(#Record) <> TypeOfElements(#Database) THEN
           RETURN;
       END_IF;
   END_REGION

   REGION Puch Record
       #_RetVal := MOVE_BLK_VARIANT(SRC := #Record, COUNT := 1, SRC_INDEX := 0, DEST_INDEX := UDINT_TO_DINT(#Act_Rec), DEST => #Database);
       IF #_RetVal = 16#0 THEN
           #Act_Rec := #Act_Rec + UDINT#1;
           #Done := TRUE;
       END_IF;
   END_REGION
END_FUNCTION

FUNCTION "fc_PopDB" : Void   // FC112, SCL
{ S7_Optimized_Access := 'TRUE' }
VERSION : 0.1
   VAR_INPUT
      Database : Variant;
      DummyRecord : Variant;
   END_VAR
   VAR_OUTPUT
      Done : Bool;
      Record : Variant;
   END_VAR
   VAR_IN_OUT
      Act_Rec : UDInt;
      Start : Bool;
   END_VAR
   VAR_TEMP
      _RecordLen : DInt;
      _Counter : DInt;
      _RetVal : Int;
      _SerializeArray : Array[1.."c_MAX_RECORD_LEN"] of Byte;
   END_VAR
BEGIN
   REGION NOT #Done
       #Done := FALSE;
   END_REGION

   REGION #Start
       IF #Start THEN
           #Start := FALSE;
       ELSE
           RETURN;
       END_IF;
   END_REGION

   REGION Check Database
       IF NOT IS_ARRAY(#Database) THEN
           RETURN;
       END_IF;
       IF #Act_Rec < UDINT#1 THEN
           RETURN;
       END_IF;
   END_REGION

   REGION Check Record
       IF (TypeOf(#Record) <> TypeOfElements(#Database)) OR (TypeOf(#Record) <> TypeOf(#DummyRecord)) THEN
           RETURN;
       END_IF;
   END_REGION

   REGION Return deleted Record
       #_RetVal := MOVE_BLK_VARIANT(SRC := #Database, COUNT := 1, SRC_INDEX := UDINT_TO_DINT(#Act_Rec -1), DEST_INDEX := 0, DEST => #Record);
   END_REGION

   REGION Prepare record with "16#0" and copy to last Record in Database
       "fc_FILL_STRUCT"(ByVAL := 16#0,
                       Struct := #DummyRecord);

       #_RetVal := MOVE_BLK_VARIANT(SRC := #DummyRecord, COUNT := 1, SRC_INDEX := 0, DEST_INDEX := UDINT_TO_DINT(#Act_Rec - 1), DEST => #Database);
       IF #_RetVal = 16#0 THEN
           #Act_Rec := #Act_Rec - UDINT#1;
           #Done := TRUE;
       END_IF;
   END_REGION
END_FUNCTION

FUNCTION "fc_ShiftDB" : Void   // FC113, SCL
{ S7_Optimized_Access := 'TRUE' }
VERSION : 0.1
   VAR_INPUT
      Database : Variant;
      DummyRecord : Variant;
   END_VAR
   VAR_OUTPUT
      Done : Bool;
      Record : Variant;
   END_VAR
   VAR_IN_OUT
      Act_Rec : UDInt;
      Start : Bool;
   END_VAR
   VAR_TEMP
      _RecordLen : DInt;
      _Counter : DInt;
      _RetVal : Int;
      _SerializeArray : Array[1.."c_MAX_RECORD_LEN"] of Byte;
   END_VAR
BEGIN
   REGION NOT #Done
       #Done := FALSE;
   END_REGION

   REGION #Start
       IF #Start THEN
           #Start := FALSE;
       ELSE
           RETURN;
       END_IF;
   END_REGION

   REGION Check Database
       IF NOT IS_ARRAY(#Database) THEN
           RETURN;
       END_IF;
       IF #Act_Rec < UDINT#1 THEN
           RETURN;
       END_IF;
   END_REGION

   REGION Check Record
       IF (TypeOf(#Record) <> TypeOfElements(#Database)) OR (TypeOf(#Record) <> TypeOf(#DummyRecord)) THEN
           RETURN;
       END_IF;
   END_REGION

   REGION Return deleted Record
       #_RetVal := MOVE_BLK_VARIANT(SRC := #Database, COUNT := 1, SRC_INDEX := 0, DEST_INDEX := 0, DEST => #Record);
       IF #_RetVal <> 16#0 THEN
           RETURN;
       END_IF;
   END_REGION

   REGION Move rest records by -1
       FOR #_Counter := DINT#2 TO UDINT_TO_DINT(#Act_Rec) DO
           #_RetVal := MOVE_BLK_VARIANT(SRC := #Database, COUNT := 1, SRC_INDEX := #_Counter - 1, DEST_INDEX := #_Counter - 2, DEST => #Database);
           IF #_RetVal <> 16#0 THEN
               RETURN;
           END_IF;
       END_FOR;
   END_REGION

   REGION Prepare record with "16#0" and copy to last Record in Database
       "fc_FILL_STRUCT"(ByVAL := 16#0,
                        Struct := #DummyRecord);
       #_RetVal := MOVE_BLK_VARIANT(SRC := #DummyRecord, COUNT := 1, SRC_INDEX := 0, DEST_INDEX := UDINT_TO_DINT(#Act_Rec - 1), DEST => #Database);
       IF #_RetVal = 0 THEN
           #Act_Rec := #Act_Rec - UDINT#1;
           #Done := TRUE;
       END_IF;
   END_REGION
END_FUNCTION

FUNCTION "fc_UnshiftDB" : Void   // FC114, SCL
{ S7_Optimized_Access := 'TRUE' }
VERSION : 0.1
   VAR_INPUT
      Record : Variant;
      Database : Variant;
   END_VAR
   VAR_OUTPUT
      Done : Bool;
   END_VAR
   VAR_IN_OUT
      Act_Rec : UDInt;
      Start : Bool;
   END_VAR
   VAR_TEMP
      _CountElements : UDInt;
      _Counter : DInt;
      _RetVal : Int;
   END_VAR
BEGIN
   REGION NOT #Done
       #Done := FALSE;
   END_REGION

   REGION #Start
       IF #Start THEN
           #Start := FALSE;
       ELSE
           RETURN;
       END_IF;
   END_REGION

   REGION Check Database
       IF IS_ARRAY(#Database) THEN
           #_CountElements := CountOfElements(#Database);
       ELSE
           RETURN;
       END_IF;
       IF #Act_Rec >=#_CountElements THEN
           RETURN;
       END_IF;
   END_REGION

   REGION Check Record
       IF TypeOf(#Record) <> TypeOfElements(#Database) THEN
           RETURN;
       END_IF;
   END_REGION

   REGION Move records by 1
       FOR #_Counter := UDINT_TO_DINT(#Act_Rec) TO DINT#1 BY DINT#-1 DO
           #_RetVal := MOVE_BLK_VARIANT(SRC := #Database, COUNT := 1, SRC_INDEX := #_Counter - 1, DEST_INDEX := #_Counter, DEST => #Database);
           IF #_RetVal <> 16#0 THEN
               RETURN;
           END_IF;
       END_FOR;
   END_REGION

   REGION Insert record at first index
       #_RetVal := MOVE_BLK_VARIANT(SRC := #Record, COUNT := 1, SRC_INDEX := 0, DEST_INDEX := 0, DEST => #Database);
       IF #_RetVal = 16#0 THEN
           #Act_Rec := #Act_Rec + UDINT#1;
           #Done := TRUE;
       END_IF;
   END_REGION
END_FUNCTION

FUNCTION "fc_ClearDB" : Void   // FC115, SCL
{ S7_Optimized_Access := 'TRUE' }
VERSION : 0.1
   VAR_INPUT
      Database : Variant;
      DummyRecord : Variant;
   END_VAR
   VAR_OUTPUT
      Done : Bool;
   END_VAR
   VAR_IN_OUT
      Act_Rec : UDInt;
      Start : Bool;
   END_VAR
   VAR_TEMP
      _CountElements : UDInt;
      _RecordLen : DInt;
      _Counter : DInt;
      _RetVal : Int;
      _SerializeArray : Array[1.."c_MAX_RECORD_LEN"] of Byte;
   END_VAR
BEGIN
   REGION NOT #Done
       #Done := FALSE;
   END_REGION

   REGION #Start
       IF #Start THEN
           #Start := FALSE;
       ELSE
           RETURN;
       END_IF;
   END_REGION

   REGION Check Database
       IF IS_ARRAY(#Database) THEN
           #_CountElements := CountOfElements(#Database);
       ELSE
           RETURN;
       END_IF;
   END_REGION

   REGION Check Record
       IF TypeOf(#DummyRecord) <> TypeOfElements(#Database) THEN
           RETURN;
       END_IF;
   END_REGION

   REGION Prepare record with "16#0" and fill whole Database
       "fc_FILL_STRUCT"(ByVAL := 16#0,
                        Struct := #DummyRecord);
       FOR #_Counter := DINT#0 TO UDINT_TO_DINT(#_CountElements - UDINT#1) DO
           #_RetVal := MOVE_BLK_VARIANT(SRC := #DummyRecord, COUNT := 1, SRC_INDEX := 0, DEST_INDEX := #_Counter, DEST => #Database);
           IF #_RetVal <> 16#0 THEN
               RETURN;
           END_IF;
       END_FOR;
       IF #_RetVal = 16#0 THEN
           #Act_Rec := UDINT#0;
       END_IF;
   END_REGION
END_FUNCTION

FUNCTION "fc_InsertDB" : Void   // FC116, SCL
{ S7_Optimized_Access := 'TRUE' }
VERSION : 0.1
   VAR_INPUT
      Record : Variant;
      Database : Variant;
      Index : UDInt;
   END_VAR
   VAR_OUTPUT
      Done : Bool;
   END_VAR
   VAR_IN_OUT
      Act_Rec : UDInt;
      Start : Bool;
   END_VAR
   VAR_TEMP
      _CountElements : UDInt;
      _Counter : DInt;
      _RetVal : Int;
   END_VAR
BEGIN
   REGION NOT #Done
       #Done := FALSE;
   END_REGION

   REGION #Start
       IF #Start THEN
           #Start := FALSE;
       ELSE
           RETURN;
       END_IF;
   END_REGION

   REGION Check Database
       IF IS_ARRAY(#Database) THEN
           #_CountElements := CountOfElements(#Database);
       ELSE
           RETURN;
       END_IF;
       IF #Act_Rec >= #_CountElements THEN
           RETURN;
       END_IF;
   END_REGION

   REGION Check Index
       IF (#Index > #Act_Rec) OR (#Index < UDINT#1) THEN
           RETURN;
       END_IF;
   END_REGION

   REGION Check Record
       IF TypeOf(#Record) <> TypeOfElements(#Database) THEN
           RETURN;
       END_IF;
   END_REGION

   REGION Move records from Index position by 1
       FOR #_Counter := UDINT_TO_DINT(#Act_Rec) TO UDINT_TO_DINT(#Index) BY DINT#-1 DO
           #_RetVal := MOVE_BLK_VARIANT(SRC := #Database, COUNT := 1, SRC_INDEX := #_Counter - 1, DEST_INDEX := #_Counter, DEST => #Database);
           IF #_RetVal <> 16#0 THEN
               RETURN;
           END_IF;
       END_FOR;
   END_REGION

   REGION Insert Record at desired Index
       #_RetVal := MOVE_BLK_VARIANT(SRC := #Record, COUNT := 1, SRC_INDEX := 0, DEST_INDEX := UDINT_TO_DINT(#Index - 1), DEST => #Database);
       IF #_RetVal = 16#0 THEN
           #Act_Rec := #Act_Rec + UDINT#1;
           #Done := TRUE;
       END_IF;
   END_REGION
END_FUNCTION

FUNCTION "fc_RemoveDB" : Void   // FC117, SCL
{ S7_Optimized_Access := 'TRUE' }
VERSION : 0.1
   VAR_INPUT
      Database : Variant;
      DummyRecord : Variant;
      Index : UDInt;
   END_VAR
   VAR_OUTPUT
      Done : Bool;
      Record : Variant;
   END_VAR
   VAR_IN_OUT
      Act_Rec : UDInt;
      Start : Bool;
   END_VAR
   VAR_TEMP
      _RecordLen : DInt;
      _Counter : DInt;
      _RetVal : Int;
      _SerializeArray : Array[1.."c_MAX_RECORD_LEN"] of Byte;
   END_VAR
BEGIN
   REGION NOT #Done
       #Done := FALSE;
   END_REGION

   REGION #Start
       IF #Start THEN
           #Start := FALSE;
       ELSE
           RETURN;
       END_IF;
   END_REGION

   REGION Check Database
       IF NOT IS_ARRAY(#Database) THEN
           RETURN;
       END_IF;
       IF #Act_Rec < UDINT#1 THEN
           RETURN;
       END_IF;
   END_REGION

   REGION Check Index
       IF (#Index > #Act_Rec) OR (#Index < UDINT#1) THEN
           RETURN;
       END_IF;
   END_REGION

   REGION Check Record
       IF (TypeOf(#Record) <> TypeOfElements(#Database)) OR (TypeOf(#Record) <> TypeOf(#DummyRecord)) THEN
           RETURN;
       END_IF;
   END_REGION

   REGION Return deleted Record
       #_RetVal := MOVE_BLK_VARIANT(SRC := #Database, COUNT := 1, SRC_INDEX := UDINT_TO_DINT(#Index - 1), DEST_INDEX := 0, DEST => #Record);
       IF #_RetVal <> 16#0 THEN
           RETURN;
       END_IF;
   END_REGION

   REGION Move rest records by -1
       FOR #_Counter := UDINT_TO_DINT(#Index) TO UDINT_TO_DINT(#Act_Rec) DO
           #_RetVal := MOVE_BLK_VARIANT(SRC := #Database, COUNT := 1, SRC_INDEX := #_Counter, DEST_INDEX := #_Counter - 1, DEST => #Database);
           IF #_RetVal <> 16#0 THEN
               RETURN;
           END_IF;
       END_FOR;
   END_REGION

   REGION Prepare record with "16#0" and copy to last Record in Database
       "fc_FILL_STRUCT"(ByVAL := 16#0,
                        Struct := #DummyRecord);
       #_RetVal := MOVE_BLK_VARIANT(SRC := #DummyRecord, COUNT := 1, SRC_INDEX := 0, DEST_INDEX := UDINT_TO_DINT(#Act_Rec - 1), DEST => #Database);
       IF #_RetVal = 0 THEN
           #Act_Rec := #Act_Rec - UDINT#1;
           #Done := TRUE;
       END_IF;
   END_REGION
END_FUNCTION

FUNCTION "fc_ReadDB" : Void   // FC118, SCL
{ S7_Optimized_Access := 'TRUE' }
VERSION : 0.1
   VAR_INPUT
      Database : Variant;
      Index : UDInt;
   END_VAR
   VAR_OUTPUT
      Done : Bool;
      Record : Variant;
   END_VAR
   VAR_IN_OUT
      Act_Rec : UDInt;
      Start : Bool;
   END_VAR
   VAR_TEMP
      _RetVal : Int;
   END_VAR
BEGIN
   REGION NOT #Done
       #Done := FALSE;
   END_REGION

   REGION #Start
       IF #Start THEN
           #Start := FALSE;
       ELSE
           RETURN;
       END_IF;
   END_REGION

   REGION Check Database
       IF NOT IS_ARRAY(#Database) THEN
           RETURN;
       END_IF;
       IF #Act_Rec <= 0 THEN
           RETURN;
       END_IF;
   END_REGION

   REGION Check Index
       IF (#Index <= UDINT#0) OR (#Index > #Act_Rec) THEN
           RETURN;
       END_IF;
   END_REGION

   REGION Check Record
       IF TypeOf(#Record) <> TypeOfElements(#Database) THEN
           RETURN;
       END_IF;
   END_REGION

   REGION Read Record
       #_RetVal := MOVE_BLK_VARIANT(SRC := #Database, COUNT := 1, SRC_INDEX := UDINT_TO_DINT(#Index - UDINT#1), DEST_INDEX := 0, DEST => #Record);
       IF #_RetVal = 16#0 THEN
           #Done := TRUE;
       END_IF;
   END_REGION
END_FUNCTION

FUNCTION "fc_ReadLastDB" : Void   // FC119, SCL
{ S7_Optimized_Access := 'TRUE' }
VERSION : 0.1
   VAR_INPUT
      Database : Variant;
   END_VAR
   VAR_OUTPUT
      Done : Bool;
      Record : Variant;
   END_VAR
   VAR_IN_OUT
      Act_Rec : UDInt;
      Start : Bool;
   END_VAR
   VAR_TEMP
      _RetVal : Int;
   END_VAR
BEGIN
   REGION NOT #Done
       #Done := FALSE;
   END_REGION

   REGION #Start
       IF #Start THEN
           #Start := FALSE;
       ELSE
           RETURN;
       END_IF;
   END_REGION

   REGION Check Database
       IF NOT IS_ARRAY(#Database) THEN
           RETURN;
       END_IF;
       IF #Act_Rec <= 0 THEN
           RETURN;
       END_IF;
   END_REGION

   REGION Check Record
       IF TypeOf(#Record) <> TypeOfElements(#Database) THEN
           RETURN;
       END_IF;
   END_REGION

   REGION Read Record
       #_RetVal := MOVE_BLK_VARIANT(SRC := #Database, COUNT := 1, SRC_INDEX := UDINT_TO_DINT(#Act_Rec - UDINT#1), DEST_INDEX := 0, DEST => #Record);
       IF #_RetVal = 16#0 THEN
           #Done := TRUE;
       END_IF;
   END_REGION
END_FUNCTION

FUNCTION "fc_OverwriteDB" : Void   // FC120, SCL
{ S7_Optimized_Access := 'TRUE' }
VERSION : 0.1
   VAR_INPUT
      Record : Variant;
      Database : Variant;
      Index : UDInt;
   END_VAR
   VAR_OUTPUT
      Done : Bool;
   END_VAR
   VAR_IN_OUT
      Act_Rec : UDInt;
      Start : Bool;
   END_VAR
   VAR_TEMP
      _RetVal : Int;
   END_VAR
BEGIN
   REGION NOT #Done
       #Done := FALSE;
   END_REGION

   REGION #Start
       IF #Start THEN
           #Start := FALSE;
       ELSE
           RETURN;
       END_IF;
   END_REGION

   REGION Check Database
       IF NOT IS_ARRAY(#Database) THEN
           RETURN;
       END_IF;
   END_REGION

   REGION Check Index
       IF (#Index > #Act_Rec) OR (#Index < UDINT#1) THEN
           RETURN;
       END_IF;
   END_REGION

   REGION Check Record
       IF TypeOf(#Record) <> TypeOfElements(#Database) THEN
           RETURN;
       END_IF;
   END_REGION

   REGION Overwrite Record at desired Index
       #_RetVal := MOVE_BLK_VARIANT(SRC := #Record, COUNT := 1, SRC_INDEX := 0, DEST_INDEX := UDINT_TO_DINT(#Index - 1), DEST => #Database);
       IF #_RetVal = 16#0 THEN
           #Done := TRUE;
       END_IF;
   END_REGION
END_FUNCTION

FUNCTION "fc_OverwriteLastDB" : Void   // FC121, SCL
{ S7_Optimized_Access := 'TRUE' }
VERSION : 0.1
   VAR_INPUT
      Record : Variant;
      Database : Variant;
   END_VAR
   VAR_OUTPUT
      Done : Bool;
   END_VAR
   VAR_IN_OUT
      Act_Rec : UDInt;
      Start : Bool;
   END_VAR
   VAR_TEMP
      _RetVal : Int;
   END_VAR
BEGIN
   REGION NOT #Done
       #Done := FALSE;
   END_REGION

   REGION #Start
       IF #Start THEN
           #Start := FALSE;
       ELSE
           RETURN;
       END_IF;
   END_REGION

   REGION Check Database
       IF NOT IS_ARRAY(#Database) THEN
           RETURN;
       END_IF;
       IF #Act_Rec <= UDINT#0 THEN
           RETURN;
       END_IF;
   END_REGION

   REGION Check Record
       IF TypeOf(#Record) <> TypeOfElements(#Database) THEN
           RETURN;
       END_IF;
   END_REGION

   REGION Overwrite Record at last Index
       #_RetVal := MOVE_BLK_VARIANT(SRC := #Record, COUNT := 1, SRC_INDEX := 0, DEST_INDEX := UDINT_TO_DINT(#Act_Rec - 1), DEST => #Database);
       IF #_RetVal = 16#0 THEN
           #Done := TRUE;
       END_IF;
   END_REGION
END_FUNCTION

FUNCTION "fc_FindDB" : Void   // FC122, SCL
{ S7_Optimized_Access := 'TRUE' }
VERSION : 0.1
   VAR_INPUT
      Record : Variant;
      RecordMask : Variant;
      Database : Variant;
   END_VAR
   VAR_OUTPUT
      Found : Bool;
      Index : UDInt;
   END_VAR
   VAR_IN_OUT
      Act_Rec : UDInt;
      TempRecord : Variant;
      Start : Bool;
   END_VAR
   VAR_TEMP
      _SerializeRecord : Array[1.."c_MAX_RECORD_LEN"] of Byte;
      _SerializeMask : Array[1.."c_MAX_RECORD_LEN"] of Byte;
      _SerializeDatabaseRecord : Array[1.."c_MAX_RECORD_LEN"] of Byte;
      _CounterRecords : UDInt;
      _CounterBytes : DInt;
      _RecordLen : DInt;
      _IndexMemo : UDInt;
      _RetVal : Int;
      _Found : Bool;
   END_VAR
BEGIN
   REGION Init
       #Found := FALSE;
       #_Found := FALSE;
       #Index := UDINT#0;
       #_IndexMemo := UDINT#0;
       #_RecordLen := DINT#0;
   END_REGION

   REGION #Start
       IF #Start THEN
           #Start := FALSE;
       ELSE
           RETURN;
       END_IF;
   END_REGION

   REGION Check Database
       IF NOT IS_ARRAY(#Database) THEN
           RETURN;
       END_IF;
       IF #Act_Rec <= UDINT#0 THEN
           RETURN;
       END_IF;
   END_REGION

   REGION Check Record
       IF (TypeOf(#Record) <> TypeOfElements(#Database)) OR (TypeOf(#Record) <> TypeOf(#RecordMask)) OR (TypeOf(#Record) <> TypeOf(#TempRecord)) THEN
           RETURN;
       END_IF;
   END_REGION

   REGION Serialize Record and RecordMask
       #_RetVal := Serialize(SRC_VARIABLE := #Record, DEST_ARRAY => #_SerializeRecord, POS := #_RecordLen);
       IF #_RetVal <> 16#0 THEN
           RETURN;
       END_IF;
       #_RecordLen := DINT#0;
       #_RetVal := Serialize(SRC_VARIABLE := #RecordMask, DEST_ARRAY => #_SerializeMask, POS := #_RecordLen);
       IF #_RetVal <> 16#0 THEN
           RETURN;
       END_IF;
   END_REGION

   REGION Compare Byte by Byte
       FOR #_CounterRecords := UDINT#1 TO #Act_Rec DO
           #_RetVal := MOVE_BLK_VARIANT(SRC := #Database, COUNT := UDINT#1, SRC_INDEX := UDINT_TO_DINT(#_CounterRecords - 1), DEST_INDEX := 0, DEST => #TempRecord);
           IF #_RetVal <> 16#0 THEN
               RETURN;
           END_IF;
           #_RecordLen := DINT#0;
           #_RetVal := Serialize(SRC_VARIABLE := #TempRecord, DEST_ARRAY => #_SerializeDatabaseRecord, POS := #_RecordLen);
           IF #_RetVal <> 16#0 THEN
               RETURN;
           END_IF;
           FOR #_CounterBytes := DINT#1 TO #_RecordLen DO
               IF (#_SerializeRecord[#_CounterBytes] <> #_SerializeDatabaseRecord[#_CounterBytes]) AND (#_SerializeMask[#_CounterBytes] = 16#FF) THEN
                   EXIT;
               END_IF;
               IF #_CounterBytes = #_RecordLen THEN
                   #_Found := TRUE;
               END_IF;
           END_FOR;
           IF #_Found THEN
               #_IndexMemo := #_CounterRecords;
               EXIT;
           END_IF;
       END_FOR;
       IF #_Found THEN
           #Found := TRUE;
           #Index := #_IndexMemo;
       END_IF;
   END_REGION
END_FUNCTION

// folder: TOOLS

FUNCTION "fc_FILL_STRUCT" : Void   // FC201, SCL
{ S7_Optimized_Access := 'TRUE' }
VERSION : 0.1
   VAR_INPUT
      ByVAL : Byte;
      "Struct" : Variant;
   END_VAR
   VAR_TEMP
      _Counter : DInt;
      _RetVal : Int;
      _SerializeArray : Array[1.."c_MAX_RECORD_LEN"] of Byte;
      _RecordLen : DInt;
   END_VAR
BEGIN
       #_RecordLen := DINT#0;
       #_RetVal := Serialize(SRC_VARIABLE := #Struct, DEST_ARRAY => #_SerializeArray, POS := #_RecordLen);
       FOR #_Counter := DINT#1 TO #_RecordLen DO
           #_SerializeArray[#_Counter] := #ByVAL;
       END_FOR;
       #_RecordLen := DINT#0;
       #_RetVal := Deserialize(SRC_ARRAY := #_SerializeArray, DEST_VARIABLE => #Struct, POS := #_RecordLen);
END_FUNCTION

FUNCTION "fc_STRING_TO_A_CHAR" : Void   // FC202, SCL
{ S7_Optimized_Access := 'TRUE' }
VERSION : 0.1
   VAR_INPUT
      IN_STRING : String;
   END_VAR
   VAR_OUTPUT
      OUT_A_Char : Variant;
   END_VAR
   VAR_TEMP
      _StringLen : DInt;
      _ArrayLen : UDInt;
      _RetVal : Int;
      _Counter : UDInt;
      _SerializeString : Array[1..256] of Char;
      _DeserializeArray : Array[1..256] of Char;
   END_VAR
BEGIN
   IF IS_ARRAY(#OUT_A_Char) THEN
       IF TypeOfElements(#OUT_A_Char) = Char THEN
           #_ArrayLen :=  CountOfElements(#OUT_A_Char);
       ELSE
           RETURN;
       END_IF;
   ELSE
       RETURN;
   END_IF;

   #_StringLen := DINT#0;
   #_RetVal := Serialize(SRC_VARIABLE := #IN_STRING, DEST_ARRAY => #_SerializeString, POS := #_StringLen);

   #_StringLen := BYTE_TO_DINT(#_SerializeString[2]);
   FOR #_Counter := UDINT#1 TO #_ArrayLen DO
       IF #_Counter <= DINT_TO_UDINT(#_StringLen) THEN
           #_DeserializeArray[#_Counter] := #_SerializeString[#_Counter + 2];
       ELSE
           #_DeserializeArray[#_Counter] := ' ';
       END_IF;
   END_FOR;

   #_StringLen := DINT#0;
   #_RetVal := Deserialize(SRC_ARRAY := #_DeserializeArray, DEST_VARIABLE => #OUT_A_Char, POS := #_StringLen);
END_FUNCTION

FUNCTION "fc_A_CHAR_TO_STRING" : Void   // FC203, SCL
{ S7_Optimized_Access := 'TRUE' }
VERSION : 0.1
   VAR_INPUT
      IN_A_CHAR : Array[*] of Char;
   END_VAR
   VAR_OUTPUT
      OUT_STRING : Variant;
   END_VAR
   VAR_TEMP
      _ArrayLo : DInt;
      _ArrayHi : DInt;
      _ArrayLen : DInt;
      _SerializeArray : Array[1..256] of Byte;
      _SerializeString : Array[1..256] of Byte;
      _Counter : DInt;
      _StringLen : DInt;
      _Factor : DInt;
      _RetVal : Int;
   END_VAR
BEGIN
   IF TypeOf(#OUT_STRING) <> String THEN
       RETURN;
   END_IF;

   #_StringLen := DINT#0;
   #_RetVal := Serialize(SRC_VARIABLE := #OUT_STRING, DEST_ARRAY => #_SerializeString, POS := #_StringLen);

   #_ArrayLo := LOWER_BOUND(ARR := #IN_A_CHAR, DIM := UDINT#1);
   #_ArrayHi := UPPER_BOUND(ARR := #IN_A_CHAR, DIM := UDINT#1);
   IF #_ArrayHi > DINT#254 THEN
       #_ArrayHi := DINT#254;
   END_IF;

   #_ArrayLen := (#_ArrayHi - #_ArrayLo) + DINT#1;
   IF #_ArrayLen > BYTE_TO_DINT(#_SerializeString[1]) THEN
       #_ArrayLen := BYTE_TO_DINT(#_SerializeString[1]);
   END_IF;

   #_Factor := #_ArrayLo - DINT#1;

   #_SerializeArray[1] := #_SerializeString[1];
   #_SerializeArray[2] := DINT_TO_BYTE(#_ArrayLen);

   FOR #_Counter := (#_ArrayLo - #_Factor) TO (#_ArrayHi - #_Factor) DO
       #_SerializeArray[#_Counter + 2] := #IN_A_CHAR[#_Counter];
   END_FOR;

   #_StringLen := DINT#0;
   #_RetVal := Deserialize(SRC_ARRAY := #_SerializeArray, DEST_VARIABLE => #OUT_STRING, POS := #_StringLen);
END_FUNCTION

// ===== library types =====

// folder: LGF/3 Comperator operations

FUNCTION "LGF_CompareVariant" : Bool   // FC10005, SCL
TITLE = LGF_CompareVariant
{ S7_Optimized_Access := 'TRUE' }
AUTHOR : Siemens_Digital_Industry
FAMILY : LGF
NAME : LGF_CompareVariant
// The function compares two structured actual parameters (array, PLC data type) and outputs whether they are of the same type and have the same values.
// 
// Compare arrays or plc datatypes and their values up to a max lengh of 200 Bytes of the connected variables. If at least one value of an element is not identical --> set function result = false
// 
// Restrictions:  
// The attached structure must not include Strings  
// The attached structure can not exceed 200 bytes, because of the internal buffer size
// Die Funktion vergleicht zwei strukturierte Aktualparameter (Array, PLC-Datentyp) und gibt aus, ob sie dem gleichen Typ entsprechen und gleiche Werte haben.
// 
// Vergleich von Arrays oder PLC Datentypen mit einer Länge von maximal 200 Bytes. Sobald eines der verglichenen Bytes unterschiedlich ist, ist das Funktionsergebniss FALSE.
// 
// Einschränkungen:
// Die verschlatenen Strukturen dürfen keine `Strings` enthalten
// Die verschaltenen Strukturen dürfen eine größe von 200 Bytes nicht überschreiden wegen der Internen Nuffergröße
   VAR_OUTPUT
      error : Bool;   // FALSE: No error / TRUE: An error occurred during the execution of the FB / FALSE: Kein Fehler / TRUE: Während der Ausführung des FB ist ein Fehler aufgetreten
      status : Word;   // 16#0000-16#7FFF: Status of the FB / 16#8000-16#FFFF: Error identification (see following Table) / 16#0000-16#7FFF: Status des FB / 16#8000-16#FFFF: Fehleridentifikation (siehe folgende Tabelle)
      subFunctionStatus : Word;   // Status or return value of called FB's, FC's and system blocks / Status oder Rückgabewert von aufgerufenen FB's / FC's und Systemfunktionen
   END_VAR
   VAR_IN_OUT
      variableA : Variant;   // First comparison variable with any data type / Erste Vergleichsvariable mit beliebigen Datentyp
      variableB : Variant;   // Second comparison variable with any data type / Zweite Vergleichsvariable mit beliebigen Datentyp
   END_VAR
   VAR_TEMP
      tempVariableASize : DInt;   // Temp store length of serialized structur of `variableA` / Temp Speicher für die Länge der serialisierten Daten aus `variableA`
      tempVariableBSize : DInt;   // Temp store length of serialized of `variableB` / Temp Speicher für die Länge der serialisierten Daten aus `variableB`
      tempindex : DInt;   // Temp index to loop trough serialzed byte arrays for comparision / Temp Schleifenindex um durch das serialisierte Byte Array zu iterieren für den Vergleich
      tempVariableAToBytes : Array[0..#MAX_LENGTH] of Byte;   // Temp store for serialized structure of `variableA` / Temp Speicher für die serialisierten Daten aus `variableA`
      tempVariableBToBytes : Array[0..#MAX_LENGTH] of Byte;   // Temp store for serialized of `variableB` / Temp Speicher für die serialisierten Daten aus `variableB`
      tempSerializeRet : Word;   // Temp `serialize` result - Errorcode >= 16#8000 if function fails / Temp Ergebnis von `serialize` - Errorcode >= 16#8000 Funktionsbearbeitung Fehlerhaft
   END_VAR
   // Ret_Val : FALSE: Values of comparison variables or PLC data types are different. TRUE: Values of the comparison variables are equal and PLC data types are identical. / FALSE: Werte der Vergleichsvariablen oder PLC-Datentypen sind unterschiedlich.TRUE: Werte der Vergleichsvariablen sind gleich und PLC-Datentypen sind identisch.
   VAR CONSTANT
      STATUS_NO_ERROR : Word := 16#0000;   // Execution finished without errors / Abarbeitung ohne Fehler beendet
      ERR_INPUT_TYPES_MUST_MATCH : Word := 16#8201;   // Error, the input types must match, e.g. STRUCT / Fehler, die Eingabetypen müssen übereinstimmen, z.B. Struct
      ERR_INPUT_TYPES_LENGTH_NOT_EQUAL : Word := 16#8202;   // Error, the input types have different lengths after serialization, `subFunctionStatus` provides an indicator of the different size / Fehler, die Eingabetypen haben nach der Serialisierung unterschiedliche Längen.`subFunctionStatus` liefert einen Indikator für die unterschiedliche Länge.
      ERR_SERIALIZE_VARIABLE_A : Word := 16#8601;   // Error occured while serialize variableA into Bytearray - see `subFunctionStatus` for detailed information / Fehler während der Serialisierung von `variableA` - weitere infos in `subFunctionStatus`
      ERR_SERIALIZE_VARIABLE_B : Word := 16#8602;   // Error occured while serialize variableB into Bytearray - see `subFunctionStatus` for detailed information / Fehler während der Serialisierung von `variableB` - weitere infos in `subFunctionStatus`
      MAX_LENGTH : Int := 200;   // Max. length of PLC data structur in Bytes, defines the internal buffer size / Max. Länge der PLC Datenstruktur, definiert die größe des internen Buffers
   END_VAR
BEGIN
   REGION BLOCK INFO HEADER
     //===============================================================================
     // SIEMENS AG / (c)Copyright 2019
     //-------------------------------------------------------------------------------
     // Title:            LGF_CompareVariant
     // Comment/Function: Compare arrays or plc datatypes and their values 
     //                   up to a max lengh of 200 Bytes of the connected variables.
     //                   If at least one value of an element is not identical -->
     //                   set function result = false
     // Library/Family:   LGF (Library General Functions)
     // Author:           Siemens Digital Industry
     // Tested with:      CPU1212C DC/DC/DC FW:V4.2
     // Engineering:      TIA Portal V15.1
     // Restrictions:     The attached structure must not include Strings
     //                   The attached structure can not exceed 200 bytes,
     //                   because of the internal buffer size
     //                   --> extend: cut from type, adjust "MAX_LENGHT" constant
     //                   ENO disabled - error handling done with error and status
     // Requirements:     PLC (S7-1200 / S7-1500)
     //-------------------------------------------------------------------------------
     // Change log table:
     // Version  | Date       | Expert in charge       | Changes applied
     // 01.00.00 03.09.2015  Siemens Industry Online Support
     //                      First released version
     // 01.00.01 11.02.2015  Siemens Industry Online Support
     //                      Bug fix
     // 01.00.02 02.01.2017  Siemens Industry Online Support
     //                      Upgrade: TIA V14 Update 1
     // 01.00.03 17.08.2018  Siemens Industry Online Support
     //                      Upgrade: TIA V15 Update 2
     // 01.00.04 23.11.2018  Siemens Industry Online Support
     //                      Upgrade: TIA V15.1
     // 01.00.05 03.06.2019  Simatic Systems Support
     //                      Refactoring and performance improvment
     //                      Change error handling to status and subFctStatus
     //                      update serialize instruction
     //                      add eno handling
     // 03.00.00 23.04.2020  Simatic Systems Support
     //                      Set version to V3.0.0, harmonize the version of the whole library
     // 03.00.01 19.01.2020  Simatic Systems Support
     //                      Insert documentation
     //===============================================================================
   END_REGION BLOCK INFO HEADER

   REGION DESCRIPTION
     (/*NOTE
   :    The status of called commands is output in `subFunctionStatus`. In this case, the output value in `status` indicates which command caused the error. In this case, refer to the TIA Portal Online Help section for information on the respective commands.

   ---

   This block compares two (structured) actual parameters and shows whether they equate to the same value.

   Note
   :    The following differences cannot be detected with the comparison method (byte level):
   * Variables of the data type `Struct` cannot be compared.
   * For strings, there may be differences in the range between the actual length and the maximum length.
   * With `REAL` numbers in the structure, a disparity can also be displayed for "same" variables.
   * Variables of the type `ARRAY of BOOL` cannot be checked for equality with the function, because the command used, `CountOfElements`, also counts the filling elements (e.g. 8 is returned with an `ARRAY[0..1] of BOOL`).
   Hinweis
   :    In `subFunctionStatus` wird der Status von aufgerufenen Anweisungen ausge-geben. Der Ausgangswert in `status` gibt in diesem Fall an, welche Anweisung den Fehler verursacht hat. Holen Sie sich in diesem Fall die Informationen aus der TIA Portal Online Hilfe zu den jeweiligen Anweisungen.

   ---

   Dieser Baustein vergleicht zwei (strukturierte) Aktualparameter und gibt aus, ob sie dem gleichen Wert entsprechen.

   Hinweis
   :    Folgende Unterschiede können mit der Vergleichsmethode (Bytelevel) nicht erkannt werden:
   * Variablen vom Datentyp `Struct` können nicht verglichen werden.
   * Bei Strings können im Bereich zwischen tatsächlicher Länge und Maximallänge Unterschiede vorhanden sein.
   * Bei `REAL` Zahlen in der Struktur kann auch bei "gleichen" Variablen eine Ungleichheit angezeigt werden.
   * Variablen vom Typ `ARRAY of BOOL` können mit der Funktion nicht auf Gleichheit geprüft werden, da die verwendete Anweisung `CountOfElements` auch die Füllelemente mitzählt (z.B. bei einem `ARRAY[0..1] of BOOL` wird 8 zurückgegeben).*/)
   END_REGION DESCRIPTION

   REGION Initialisation
     // init temporary variables
     #tempVariableASize := 0;
     #tempVariableBSize := 0;
     #tempindex := 0;

     // Set "No current job" #status
     #error := FALSE;
     #status := #STATUS_NO_ERROR;
     #subFunctionStatus := #STATUS_NO_ERROR;

     // Initialisation of function result
     #LGF_CompareVariant := FALSE;
   END_REGION Initialisation

   REGION Processing

     REGION Check input types
       // Check if the datatypes of the connected tags are identical
       IF TypeOf(#variableA) <> TypeOf(#variableB) THEN
         #error := TRUE;
         #status := #ERR_INPUT_TYPES_MUST_MATCH;
         #subFunctionStatus := #STATUS_NO_ERROR;
         // no error handling needed
         ENO := TRUE;
         RETURN; // Finish function if conversion fails
       END_IF;
     END_REGION

     REGION Serialize Input Variable A
       // convert variableA Values to serialised binary array of byte
       #tempSerializeRet := INT_TO_WORD(
                                        Serialize(SRC_VARIABLE := #variableA,
                                                  DEST_ARRAY => #tempVariableAToBytes,
                                                  POS := #tempVariableASize)
       );

       // Check return value of SERIALIZE
       // if not zero - error happend, write error codes and end/leave function
       IF #tempSerializeRet <> #STATUS_NO_ERROR THEN
         #error := TRUE;
         #status := #ERR_SERIALIZE_VARIABLE_A;
         #subFunctionStatus := #tempSerializeRet;
         // no error handling needed
         ENO := TRUE;
         RETURN; // Finish function if conversion fails
       END_IF;
     END_REGION

     REGION Serialize Input Variable A
       // convert variableB Values to serialised binary array of byte
       #tempSerializeRet := INT_TO_WORD(
                                        Serialize(SRC_VARIABLE := #variableB,
                                                  DEST_ARRAY => #tempVariableBToBytes,
                                                  POS := #tempVariableBSize)
       );

       // Check return value of SERIALIZE
       // if not zero - error happend, write error codes and end/leave function
       IF #tempSerializeRet <> #STATUS_NO_ERROR THEN
         #error := TRUE;
         #status := #ERR_SERIALIZE_VARIABLE_B;
         #subFunctionStatus := #tempSerializeRet;
         // no error handling needed
         ENO := TRUE;
         RETURN; // Finish function if conversion fails
       END_IF;
     END_REGION

     REGION Check if serialized sizes are equal
       // Compare size of both variables
       IF #tempVariableASize <> #tempVariableBSize THEN
         #error := TRUE;
         #status := #ERR_INPUT_TYPES_LENGTH_NOT_EQUAL;
         #subFunctionStatus := DINT_TO_WORD(#tempVariableASize - #tempVariableBSize);
         // no error handling needed
         ENO := TRUE;
         RETURN; // Finish function if conversion fails
       END_IF;
     END_REGION

     REGION Compare
       // Compare values of temp. array elements of bytes
       WHILE #tempindex < #tempVariableASize DO

         // Compare bytes till difference detected
         IF #tempVariableAToBytes[#tempindex] = #tempVariableBToBytes[#tempindex] THEN
           // if equal increment index
           #tempindex += 1; // Or end of array reached
         ELSE
           // if values diffrent (content missmatch) --> exit loop
           EXIT;
         END_IF;
       END_WHILE;

     END_REGION
   END_REGION Processing

   REGION Output
     // Assign function result - if index is equal to size = TRUE
     #LGF_CompareVariant := (#tempindex = #tempVariableASize);

     // ENO is not used, forced to TRUE
     ENO := TRUE;
   END_REGION
END_FUNCTION